{attribute 'linkalways'} 
{attribute 'no_explicit_call' := 'This FB is a CLASS and must be accessed using methods or properties'}
{attribute 'enable_dynamic_creation'}
FUNCTION_BLOCK Node_F_VN_ConvertCartesianToPolarAngles EXTENDS VisionNode
VAR
	ipSrcPointsCart : _ITcVnContainer;
    ipDestAngles : _ITcVnContainer;
    hrPrev : _HRESULT(S_OK);
	hresult : _HRESULT(S_OK);
END_VAR

METHOD PUBLIC  Clone : I_Node
VAR
	pNode : POINTER TO Node_F_VN_ConvertCartesianToPolarAngles;
END_VAR
pNode := __NEW(Node_F_VN_ConvertCartesianToPolarAngles);
Clone := pNode^;
END_METHOD

METHOD FB_init : BOOL
VAR_INPUT
	bInitRetains : BOOL; // if TRUE, the retain variables are initialized (warm start / cold start)
	bInCopyCode : BOOL;  // if TRUE, the instance afterwards gets moved into the copy code (online change)
END_VAR
AddInput('ipSrcPointsCart', ipSrcPointsCart);
AddInput('hrPrev', hrPrev);
AddOutput('ipDestAngles', ipDestAngles);
AddOutput('hresult',hresult);
END_METHOD

METHOD PROTECTED OnExecute
hresult.Value := F_VN_ConvertCartesianToPolarAngles(
	ipSrcPointsCart := ipSrcPointsCart.Value, 
	ipDestAngles := ipDestAngles.Value, 
	hrPrev := hrPrev.Value);
END_METHOD

METHOD PUBLIC PreExecutionCheck
VAR_INPUT
	Check : I_PreExecutionChecks;
END_VAR
Check.IsTrue(ipSrcPointsCart.IsValid, 'ipSrcPointsCart must be a valid container');
Check.IsTrue((ipSrcPointsCart.IsType(TC_GLOBAL_CONST_LIST.ContainerType_Vector_TcVnPoint2_DINT) OR
              ipSrcPointsCart.IsType(TC_GLOBAL_CONST_LIST.ContainerType_Vector_TcVnPoint2_REAL) OR
              ipSrcPointsCart.IsType(TC_GLOBAL_CONST_LIST.ContainerType_Vector_TcVnPoint2_LREAL)),
              'ipSrcPointsCart contains incorrect type');
END_METHOD

END_FUNCTION_BLOCK

(* stored: Version 1.1.0.1, ProductVersion 3.1.4026.13
   POU Node_F_VN_ConvertCartesianToPolarAngles: Id {2551c897-175e-0916-1cd9-9b9f150002d7}, SpecialFunc None
   Folder Constructor: Id {462c05f3-7bac-0f04-20ae-2e3732d6d174}
   Method Clone: Id {29b7c63f-03b7-03e7-2684-7ae3acd424ab}
   Method FB_init: Id {03e6c768-b066-0c8a-1281-b69ccea23afa}
   Method OnExecute: Id {eb98bf9c-8d86-0779-1181-2b319935a594}
   Method PreExecutionCheck: Id {35e6354d-4cda-00f2-0dfe-cb76188b42ef} *)
